Staubli VAL3: toggleValve.pgx

program toggleValve(num iValve)
begin
  if statusValves[iValve]==1
    statusValves[iValve]=0
    colorValveButton[iValve]=colorOff
    switch iValve
      case 0
        doJ206_EtherCAT_Box_1__CPX_FB37__Q0[0]=false
      break
      case 1
        doJ206_EtherCAT_Box_1__CPX_FB37__Q1[0]=false
      break
      case 2
        doJ206_EtherCAT_Box_1__CPX_FB37__Q2[0]=false
      break
      case 3
        doJ206_EtherCAT_Box_1__CPX_FB37__Q3[0]=false
      break
      case 4
        doJ206_EtherCAT_Box_1__CPX_FB37__Q4[0]=false
      break
      case 5
        doJ206_EtherCAT_Box_1__CPX_FB37__Q5[0]=false
      break
      case 6
        doJ206_EtherCAT_Box_1__CPX_FB37__Q6[0]=false
      break
      case 7
        doJ206_EtherCAT_Box_1__CPX_FB37__Q7[0]=false
      break
      case 8
        doJ206_EtherCAT_Box_1__CPX_FB37__Q8[0]=false
      break
      case 9
        doJ206_EtherCAT_Box_1__CPX_FB37__Q9[0]=false
      break
      case 10
        doJ206_EtherCAT_Box_1__CPX_FB37__Q10[0]=false
      break
      case 11
        doJ206_EtherCAT_Box_1__CPX_FB37__Q11[0]=false
      break
      case 12
        doJ206_EtherCAT_Box_1__CPX_FB37__Q12[0]=false
      break
      case 13
        doJ206_EtherCAT_Box_1__CPX_FB37__Q13[0]=false
      break
      case 14
        doJ206_EtherCAT_Box_1__CPX_FB37__Q14[0]=false
      break
      case 15
        doJ206_EtherCAT_Box_1__CPX_FB37__Q15[0]=false
      break
      case 16
        doJ206_EtherCAT_Box_1__CPX_FB37__Q16[0]=false
      break
      case 17
        doJ206_EtherCAT_Box_1__CPX_FB37__Q17[0]=false
      break
    endSwitch
  else
    statusValves[iValve]=1
    colorValveButton[iValve]=colorOn
    switch iValve
      case 0
        doJ206_EtherCAT_Box_1__CPX_FB37__Q0[0]=true
      break
      case 1
        doJ206_EtherCAT_Box_1__CPX_FB37__Q1[0]=true
      break
      case 2
        doJ206_EtherCAT_Box_1__CPX_FB37__Q2[0]=true
      break
      case 3
        doJ206_EtherCAT_Box_1__CPX_FB37__Q3[0]=true
      break
      case 4
        doJ206_EtherCAT_Box_1__CPX_FB37__Q4[0]=true
      break
      case 5
        doJ206_EtherCAT_Box_1__CPX_FB37__Q5[0]=true
      break
      case 6
        doJ206_EtherCAT_Box_1__CPX_FB37__Q6[0]=true
      break
      case 7
        doJ206_EtherCAT_Box_1__CPX_FB37__Q7[0]=true
      break
      case 8
        doJ206_EtherCAT_Box_1__CPX_FB37__Q8[0]=true
      break
      case 9
        doJ206_EtherCAT_Box_1__CPX_FB37__Q9[0]=true
      break
      case 10
        doJ206_EtherCAT_Box_1__CPX_FB37__Q10[0]=true
      break
      case 11
        doJ206_EtherCAT_Box_1__CPX_FB37__Q11[0]=true
      break
      case 12
        doJ206_EtherCAT_Box_1__CPX_FB37__Q12[0]=true
      break
      case 13
        doJ206_EtherCAT_Box_1__CPX_FB37__Q13[0]=true
      break
      case 14
        doJ206_EtherCAT_Box_1__CPX_FB37__Q14[0]=true
      break
      case 15
        doJ206_EtherCAT_Box_1__CPX_FB37__Q15[0]=true
      break
      case 16
        doJ206_EtherCAT_Box_1__CPX_FB37__Q16[0]=true
      break
      case 17
        doJ206_EtherCAT_Box_1__CPX_FB37__Q17[0]=true
      break
    endSwitch
  endIf

  // -- setup button colors for frontpage
  if statusValves[airexValve[0]] == 1 and statusValves[airexValve[1]] == 1  and statusValves[airexValve[2]] == 1 and  statusValves[airexValve[3]] == 1 and statusValves[airexValve[4]] == 1 and statusValves[airexValve[5]] == 1
    colorVacuumStatus1 = colorOn
  else
    colorVacuumStatus1 = colorOff
  endIf


end
